FUNCTION_BLOCK FB_ExcitationPulseModulation
VAR
	bIncrease	:	BOOL;
	bDecrease	: 	BOOL;
	
	bIncPulse	:	BOOL;
	bDecPulse	:	BOOL;
	
	iPulseWidth	:	INT;
	iNumOfPulse	:	INT;
	iDelayTime	:	INT;
	
	tonPulseCreation :	TON;
	bOutPulse	:	BOOL;
	iStep		:	INT;
	iLoop		:	INT;
	bPulse		:	BOOL;
	bDelayStep	:	BOOL := TRUE;
END_VAR

CASE iStep OF 
	0: // Wait for command
		IF bIncrease OR bDecrease THEN
			iStep := 5;
		END_IF
		
	5: // Init
		tonPulseCreation.PT := INT_TO_TIME(iPulseWidth);
		iLoop := 0;
		iStep := 10;
		
	10:	// Create pulse
		bPulse := TRUE;
		IF tonPulseCreation.Q THEN
			tonPulseCreation(IN := FALSE);
			iStep := 15;
		END_IF
		
	15: // Pulse off
		bPulse := FALSE;
		IF tonPulseCreation.Q THEN
			tonPulseCreation(IN := FALSE);
			iStep := 17;
		END_IF
		
	17: // Check loop
		IF iLoop < iNumOfPulse - 1 THEN
			iStep := 10;
			iLoop := iLoop + 1;
		ELSE
			iStep := 20;
			iLoop := 0;
			tonPulseCreation.PT := INT_TO_TIME(iDelayTime - iPulseWidth);
		END_IF
		
	20: // Delay pusle 
		bPulse := FALSE;
		IF tonPulseCreation.Q THEN
			tonPulseCreation(IN := FALSE);
			iStep := 30;
		END_IF
		
	30: // Complete
		IF NOT bIncrease AND NOT bDecrease THEN 
			iStep := 0;
		END_IF
	
END_CASE


tonPulseCreation(IN := iStep >= 10 AND iStep <= 20);

bIncPulse := bIncrease AND bPulse;
bDecPulse := bDecrease AND bPulse;

bIncrease := FALSE;
bDecrease := FALSE;

PROPERTY DecPulse : BOOL
GET
DecPulse := bDecPulse;
END_GET
END_PROPERTY

METHOD Decrease : BOOL
VAR_INPUT
END_VAR
bDecrease := TRUE;

Decrease := bDecrease AND iStep = 30;
END_METHOD

PROPERTY IncPulse : BOOL
GET
IncPulse := bIncPulse;
END_GET
END_PROPERTY

METHOD Increase : BOOL
VAR_INPUT
END_VAR
bIncrease := TRUE;

Increase := bIncrease AND iStep = 30;
END_METHOD

END_FUNCTION_BLOCK

(* stored: Version 1.1.0.1, ProductVersion 3.1.4024.12
   POU FB_ExcitationPulseModulation: Id {b8ab3866-b4ca-4583-8e82-dd7ab239c044}, SpecialFunc None
   Property DecPulse: Id {2aa10090-6c2e-4d8c-8d99-0f32b114f2ca}
   Get Get: Id {2f8d1df4-47c7-43c2-9ee9-beacd141468a}
   Method Decrease: Id {ca61c3aa-9f50-49a3-b7ef-3e4707172db9}
   Property IncPulse: Id {a81b2a3f-0397-4167-9774-d55a58dee1b4}
   Get Get: Id {b94d3f15-ac19-4edd-a405-51ba0a0b4e95}
   Method Increase: Id {b4370d50-8e0e-4df2-a00b-3f3de7551bea} *)
